# EPICS autosave request: iocBoot/sioc-esb-adps40/auto_settings.req
file "ADBase_settings.req",         P=$(P),  R=cam1:
#file "NDFile_settings.req",         P=$(P),  R=TIFF1:
file "prosilica_settings.req",      P=$(P),  R=cam1:
file "NDPluginBase_settings.req",   P=$(P),  R=image1:
file "NDStdArrays_settings.req",    P=$(P),  R=image1:
file "../prosilica.req",            P=$(P)
